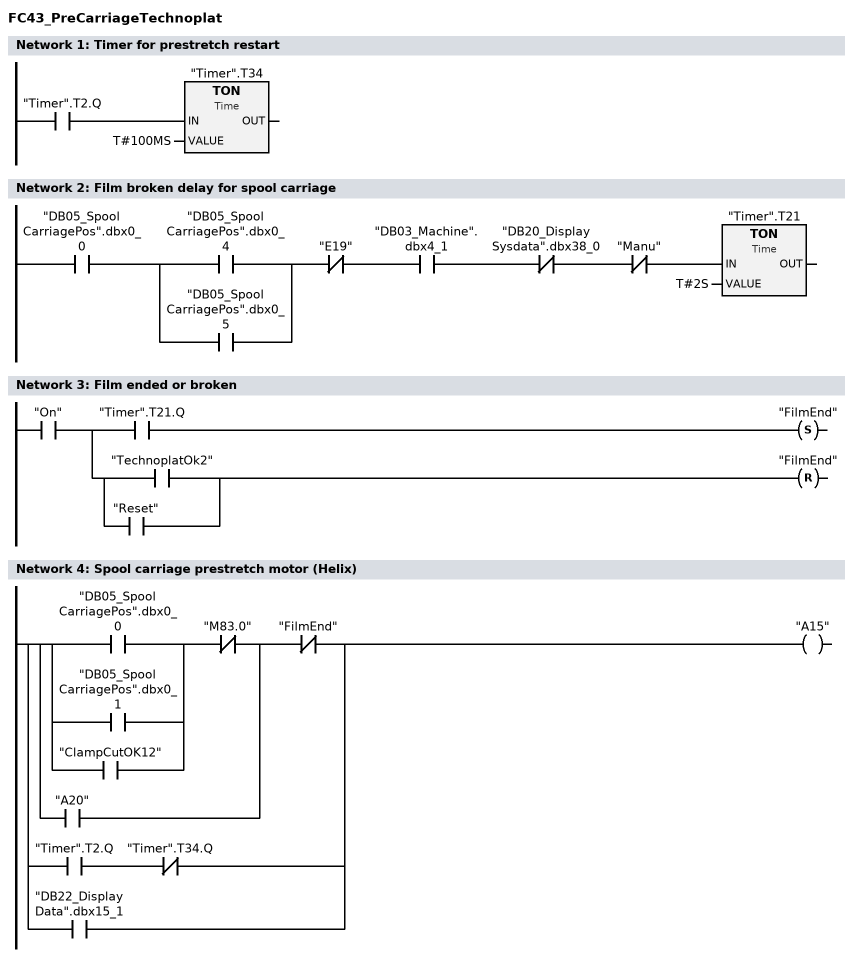
   "Timer".T34.TON(IN := "Timer".T2.Q, PT := T#100MS);   // TON coil
END_REGION

REGION Network 2: Film broken delay for spool carriage
   "Timer".T21.TON(IN := "DB05_SpoolCarriagePos".dbx0_0 AND ("DB05_SpoolCarriagePos".dbx0_4 OR "DB05_SpoolCarriagePos".dbx0_5) AND NOT "E19" AND "DB03_Machine".dbx4_1 AND NOT "DB20_DisplaySysdata".dbx38_0 AND NOT "Manu", PT := T#2S);   // TON coil
END_REGION

REGION Network 3: Film ended or broken
   RUNG wire#powerrail
      Contact( "On" )
      wire#w1
      Contact( "Timer".T21.Q )
      S_Coil( "FilmEnd" )
   END_RUNG
   RUNG wire#w1
      Contact( "TechnoplatOk2" )
      wire#w2
      R_Coil( "FilmEnd" )
   END_RUNG
   RUNG wire#w1
      Contact( "Reset" )
   END_RUNG wire#w2
   // the same network as SCL:
   IF "On" AND "Timer".T21.Q THEN "FilmEnd" := TRUE; END_IF;
   IF "On" AND ("TechnoplatOk2" OR "Reset") THEN "FilmEnd" := FALSE; END_IF;
END_REGION

REGION Network 4: Spool carriage prestretch motor (Helix)
   RUNG wire#powerrail
      Contact( "DB05_SpoolCarriagePos".dbx0_0 )
      wire#w1
      I_Contact( "M83.0" )
      wire#w2
      I_Contact( "FilmEnd" )
      wire#w3
      Coil( "A15" )
   END_RUNG
   RUNG wire#powerrail
      Contact( "DB05_SpoolCarriagePos".dbx0_1 )
   END_RUNG wire#w1
   RUNG wire#powerrail
      Contact( "ClampCutOK12" )
   END_RUNG wire#w1
   RUNG wire#powerrail
      Contact( "A20" )
   END_RUNG wire#w2
   RUNG wire#powerrail
      Contact( "Timer".T2.Q )
      I_Contact( "Timer".T34.Q )
   END_RUNG wire#w3
   RUNG wire#powerrail
      Contact( "DB22_DisplayData".dbx15_1 )
   END_RUNG wire#w3
   // the same network as SCL:
   "A15" := (((("DB05_SpoolCarriagePos".dbx0_0 OR "DB05_SpoolCarriagePos".dbx0_1 OR "ClampCutOK12") AND NOT "M83.0") OR "A20") AND NOT "FilmEnd") OR ("Timer".T2.Q AND NOT "Timer".T34.Q) OR "DB22_DisplayData".dbx15_1;
END_REGION
END_FUNCTION

FUNCTION "FC62_PreStretchPGSAoutPWM" : Void   // FC62, LAD
{ S7_Optimized_Access := 'FALSE' }
AUTHOR : PaZan
VERSION : 0.1
// stored: AutoNumber false, IsIECCheckEnabled false, SetENOAutomatically false, UDAEnableTagReadback false
BEGIN

REGION Network 1: copy parameter for scale value % prestretch
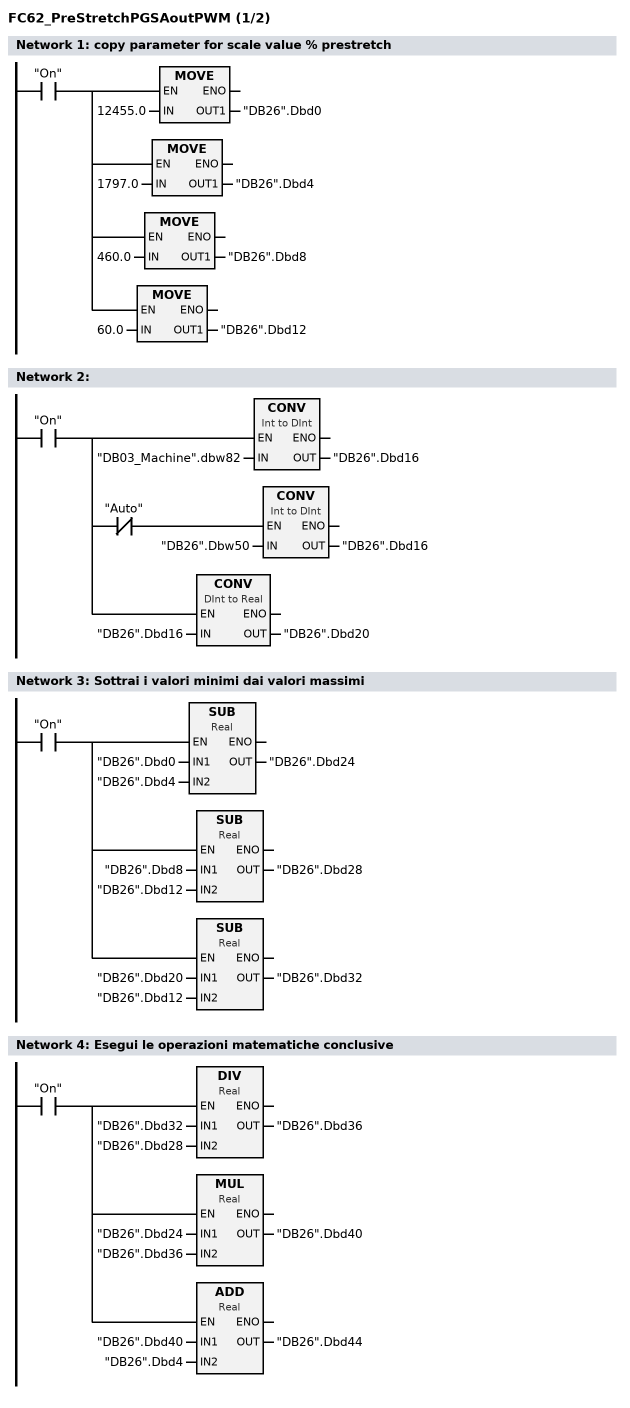
   RUNG wire#powerrail
      Contact( "On" )
      wire#w1
      { S7_GenerateENO := "TRUE" } Move(in := 12455.0, out1 => "DB26".Dbd0)
   END_RUNG
   RUNG wire#w1
      { S7_GenerateENO := "TRUE" } Move(in := 1797.0, out1 => "DB26".Dbd4)
   END_RUNG
   RUNG wire#w1
      { S7_GenerateENO := "TRUE" } Move(in := 460.0, out1 => "DB26".Dbd8)
   END_RUNG
   RUNG wire#w1
      { S7_GenerateENO := "TRUE" } Move(in := 60.0, out1 => "DB26".Dbd12)
   END_RUNG
   // the same network as SCL:
   IF "On" THEN
       "DB26".Dbd0 := 12455.0;
       "DB26".Dbd4 := 1797.0;
       "DB26".Dbd8 := 460.0;
       "DB26".Dbd12 := 60.0;
   END_IF;
END_REGION

REGION Network 2
   RUNG wire#powerrail
      Contact( "On" )
      wire#w1
      { S7_Templates := "[SrcType := Int, DestType := DInt]"; S7_GenerateENO := "TRUE" } Convert(in := "DB03_Machine".dbw82, out => "DB26".Dbd16)
   END_RUNG
   RUNG wire#w1
      I_Contact( "Auto" )
      { S7_Templates := "[SrcType := Int, DestType := DInt]"; S7_GenerateENO := "TRUE" } Convert(in := "DB26".Dbw50, out => "DB26".Dbd16)
   END_RUNG
   RUNG wire#w1
      { S7_Templates := "[SrcType := DInt, DestType := Real]"; S7_GenerateENO := "TRUE" } Convert(in := "DB26".Dbd16, out => "DB26".Dbd20)
   END_RUNG
   // the same network as SCL:
   IF "On" THEN "DB26".Dbd16 := INT_TO_DINT("DB03_Machine".dbw82); END_IF;
   IF "On" AND NOT "Auto" THEN "DB26".Dbd16 := INT_TO_DINT("DB26".Dbw50); END_IF;
   IF "On" THEN "DB26".Dbd20 := DINT_TO_REAL("DB26".Dbd16); END_IF;
END_REGION

REGION Network 3: Sottrai i valori minimi dai valori massimi
   RUNG wire#powerrail
      Contact( "On" )
      wire#w1
      { S7_Templates := "SrcType := Real"; S7_GenerateENO := "TRUE" } Sub(in1 := "DB26".Dbd0, in2 := "DB26".Dbd4, out => "DB26".Dbd24)
   END_RUNG
   RUNG wire#w1
      { S7_Templates := "SrcType := Real"; S7_GenerateENO := "TRUE" } Sub(in1 := "DB26".Dbd8, in2 := "DB26".Dbd12, out => "DB26".Dbd28)
   END_RUNG
   RUNG wire#w1
      { S7_Templates := "SrcType := Real"; S7_GenerateENO := "TRUE" } Sub(in1 := "DB26".Dbd20, in2 := "DB26".Dbd12, out => "DB26".Dbd32)
   END_RUNG
   // the same network as SCL:
   IF "On" THEN
       "DB26".Dbd24 := "DB26".Dbd0 - "DB26".Dbd4;
       "DB26".Dbd28 := "DB26".Dbd8 - "DB26".Dbd12;
       "DB26".Dbd32 := "DB26".Dbd20 - "DB26".Dbd12;
   END_IF;
END_REGION

REGION Network 4: Esegui le operazioni matematiche conclusive
   RUNG wire#powerrail
      Contact( "On" )
      wire#w1
      { S7_Templates := "SrcType := Real"; S7_GenerateENO := "TRUE" } Div(in1 := "DB26".Dbd32, in2 := "DB26".Dbd28, out => "DB26".Dbd36)
   END_RUNG
   RUNG wire#w1
      { S7_Templates := "SrcType := Real"; S7_GenerateENO := "TRUE" } Mul(in1 := "DB26".Dbd24, in2 := "DB26".Dbd36, out => "DB26".Dbd40)
   END_RUNG
   RUNG wire#w1
      { S7_Templates := "SrcType := Real"; S7_GenerateENO := "TRUE" } Add(in1 := "DB26".Dbd40, in2 := "DB26".Dbd4, out => "DB26".Dbd44)
   END_RUNG
   // the same network as SCL:
   IF "On" THEN
       "DB26".Dbd36 := "DB26".Dbd32 / "DB26".Dbd28;
       "DB26".Dbd40 := "DB26".Dbd24 * "DB26".Dbd36;
       "DB26".Dbd44 := "DB26".Dbd40 + "DB26".Dbd4;
   END_IF;
END_REGION

REGION Network 5: Trunc and copy value for pre-stretch in analogic out
   // PAW128
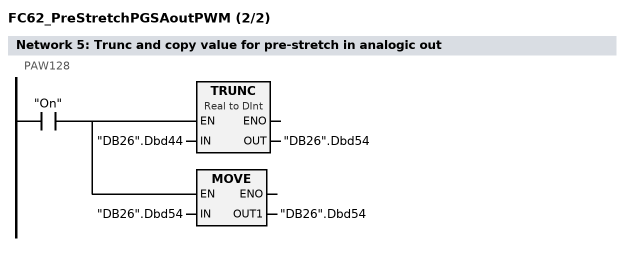
   RUNG wire#powerrail
      Contact( "On" )
      wire#w1
      { S7_Templates := "[SrcType := Real, DestType := DInt]"; S7_GenerateENO := "TRUE" } Trunc(in := "DB26".Dbd44, out => "DB26".Dbd54)
   END_RUNG
   RUNG wire#w1
      { S7_GenerateENO := "TRUE" } Move(in := "DB26".Dbd54, out1 => "DB26".Dbd54)
   END_RUNG
   // the same network as SCL:
   IF "On" THEN
       "DB26".Dbd54 := TRUNC("DB26".Dbd44);
       "DB26".Dbd54 := "DB26".Dbd54;
   END_IF;
END_REGION
END_FUNCTION

DATA_BLOCK "U201_Process_Data"   // DB211
VERSION : 0.1
// stored: AutoNumber false, InstanceOfName Inverter_Process_Data, InstanceOfType FB
"Inverter_Process_Data"
BEGIN
END_DATA_BLOCK

DATA_BLOCK "U221_Process_Data"   // DB212
VERSION : 0.1
// stored: AutoNumber false, InstanceOfName Inverter_Process_Data, InstanceOfType FB
"Inverter_Process_Data"
BEGIN
END_DATA_BLOCK
